FUNCTION_BLOCK W1W2
  (* Standard: 61499-2 *)
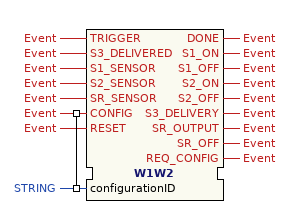
  EVENT_INPUT
    TRIGGER;
    S3_DELIVERED;
    S1_SENSOR;
    S2_SENSOR;
    SR_SENSOR;
    CONFIG WITH configurationID;
    RESET;
  END_EVENT
  EVENT_OUTPUT
    DONE;
    S1_ON;
    S1_OFF;
    S2_ON;
    S2_OFF;
    S3_DELIVERY;
    SR_OUTPUT;
    SR_OFF;
    REQ_CONFIG;
  END_EVENT
  VAR_INPUT
    configurationID : STRING;
  END_VAR
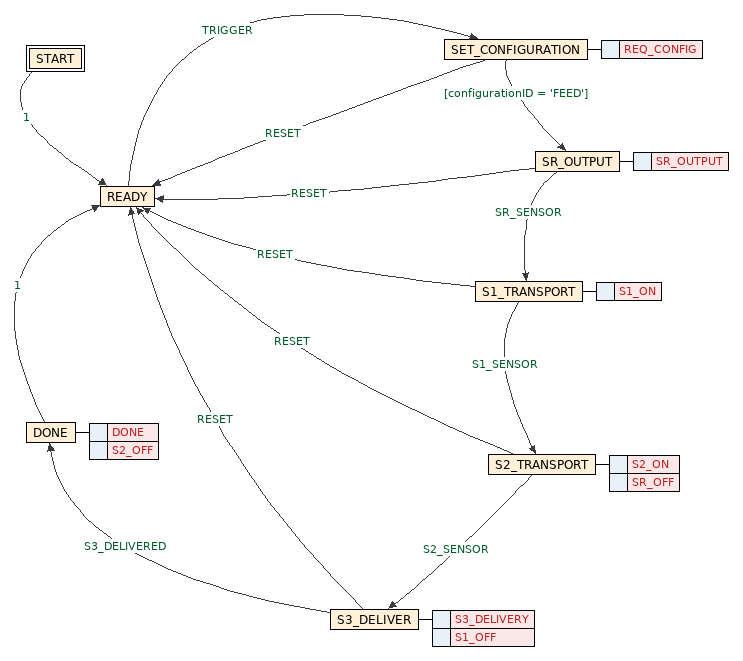
  EC_STATES
    START;
    SR_OUTPUT : -> SR_OUTPUT;
    S1_TRANSPORT : -> S1_ON;
    S2_TRANSPORT : -> S2_ON, -> SR_OFF;
    S3_DELIVER : -> S3_DELIVERY, -> S1_OFF;
    DONE : -> DONE, -> S2_OFF;
    READY;
    SET_CONFIGURATION : -> REQ_CONFIG;
  END_STATES
  EC_TRANSITIONS
    START TO READY := 1;
    SR_OUTPUT TO S1_TRANSPORT := SR_SENSOR;
    S1_TRANSPORT TO S2_TRANSPORT := S1_SENSOR;
    S2_TRANSPORT TO S3_DELIVER := S2_SENSOR;
    S3_DELIVER TO DONE := S3_DELIVERED;
    READY TO SET_CONFIGURATION := TRIGGER;
    SET_CONFIGURATION TO SR_OUTPUT := [configurationID = 'FEED'];
    DONE TO READY := 1;
    SET_CONFIGURATION TO READY := RESET;
    SR_OUTPUT TO READY := RESET;
    S1_TRANSPORT TO READY := RESET;
    S2_TRANSPORT TO READY := RESET;
    S3_DELIVER TO READY := RESET;
  END_TRANSITIONS
  ALGORITHM INIT IN ST:

  END_ALGORITHM
  ALGORITHM REQ IN ST:

  END_ALGORITHM
END_FUNCTION_BLOCK
